FUNCTION_BLOCK fbDrive
VAR
	{attribute addProperty Name "Position"}
    {attribute addProperty Units "nm"}	
	Position : LREAL;
	{attribute addProperty Name "Speed"}
	{attribute addProperty Units "mm/s"}
	Speed : LREAL;
	{attribute addProperty Name "Acceleration"}
	{attribute addProperty Units "mm/s^2"}
	Acc : REAL;
	{attribute addProperty Name "Deceleration"}
	{attribute addProperty Units "mm/s^2"}
	Dcc : REAL;
END_VAR

Position := Position + 0.1;
Speed := Position / 0.025;
Acc := 1000.0;
Dcc := 1000.0;

END_FUNCTION_BLOCK

(* stored: Version 1.1.0.1, ProductVersion 3.1.4024.2
   POU fbDrive: Id {3dc76d49-1038-4ada-b247-e6bb10b2c1e9}, SpecialFunc None *)
